INTERFACE ITFComponent EXTENDS __SYSTEM.IQueryInterface

/// Get's or set's a value indicating whether this component is active or not.
PROPERTY Active : BOOL
GET
END_GET
SET
END_SET
END_PROPERTY

PROPERTY BMK : STRING
GET
END_GET
SET
END_SET
END_PROPERTY

/// Get's value representing the component state.
PROPERTY ClearText : String
GET
END_GET
END_PROPERTY

PROPERTY ID : INT
GET
END_GET
SET
END_SET
END_PROPERTY

/// Get's value representing the component state.
PROPERTY LastError : STRING
GET
END_GET
END_PROPERTY

PROPERTY MachineArea : E_MachineArea
GET
END_GET
SET
END_SET
END_PROPERTY

PROPERTY Name : STRING
GET
END_GET
SET
END_SET
END_PROPERTY

PROPERTY Path : String
GET
END_GET
END_PROPERTY

/// Reset component logic
{attribute 'object_name' := 'Reset'}
METHOD Reset
END_METHOD

/// Run component logic
{attribute 'object_name' := 'Run'}
METHOD Run : E_ComponentState
END_METHOD

/// Set HMI reference
METHOD SetEventLogReference
VAR_IN_OUT
	/// HMI access provider.
	fbEventLogRef	: FB_EventLog;
END_VAR
END_METHOD

/// Get's value representing the component state.
PROPERTY State : E_ComponentState
GET
END_GET
END_PROPERTY

/// Get's value representing the component state.
PROPERTY StateAsString : STRING
GET
END_GET
END_PROPERTY

PROPERTY Typ : E_ComponentType
GET
END_GET
END_PROPERTY

END_INTERFACE

(* stored: Version 1.1.0.1, ProductVersion 3.1.4022.7
   Itf ITFComponent: Id {0c339870-3919-4156-9e10-4458967cc3e3}
   Property Active: Id {a4013bac-f678-40d6-b6e3-75f80b396d7b}
   Get Get: Id {b22ecde3-e151-433e-b7bb-73c02ebc3421}
   Set Set: Id {8a51a58a-f21e-40e0-b475-07986ff1617d}
   Property BMK: Id {be910f48-dfb5-41ca-90d6-b34daf26889e}
   Get Get: Id {f9e623e8-0a55-4a0a-81f8-be539998713c}
   Set Set: Id {672c2167-4352-435e-9e87-a06ddfb483ac}
   Property ClearText: Id {1b270129-2b79-4ed2-8681-18554c509971}
   Get Get: Id {0ded3386-5c43-4f6e-ab50-341431662cd6}
   Property ID: Id {d6eb581a-9300-43d2-a537-fd27c418df38}
   Get Get: Id {5ba80d43-ea9e-4854-a96a-c1d86a80c18d}
   Set Set: Id {f550cafb-024d-4181-a215-7f6db2e96e7d}
   Property LastError: Id {f1d9d119-6784-4c74-950f-734bdedcbab4}
   Get Get: Id {cff7ecae-c39e-4dbe-9014-c2be392b15d3}
   Property MachineArea: Id {92788664-5c69-4a9c-9046-f9b02a731813}
   Get Get: Id {fd4531d5-8c1b-4e7b-922e-1d59f20e9078}
   Set Set: Id {875a4e47-605d-4116-91d3-7ec864ef4f3b}
   Property Name: Id {dfe3cfb1-960f-481b-9895-7c3d2fdb66bb}
   Get Get: Id {d6a0caca-8384-434e-b687-46dd7b90c949}
   Set Set: Id {d763021b-6a1b-4ad2-8f31-f17edf192944}
   Property Path: Id {d49383b0-7900-4755-8881-e6510a11411d}
   Get Get: Id {1f792d33-338d-486d-ba2f-8947ff9e5e1c}
   Method Reset: Id {d20f6564-ac00-4f07-b6e7-4efc746c414a}
   Method Run: Id {9456d1b6-8b95-48fd-bbab-7ac1c5ad6db3}
   Method SetEventLogReference: Id {770eda9c-2cf8-49f7-85fb-b7d4677747c2}
   Property State: Id {62ee10f7-b429-4216-b697-b5f173ac2511}
   Get Get: Id {197f3a44-b9d4-40e1-8c9e-c1a1588c0941}
   Property StateAsString: Id {6b6e811f-0f6a-45c4-af3a-a9178954bbe3}
   Get Get: Id {143d593f-bcf8-40cd-99de-5c114b1299bb}
   Property Typ: Id {600151d1-2b3c-4c87-a5bb-ed8db31b21c9}
   Get Get: Id {d1fdd419-1617-479d-9337-fcd8948815ed} *)
